# EPICS autosave request: iocBoot/ioc13ida_linux/Galil_settings.req
file "CARS_32_motor_settings.req",     P=$(P)
file "CARS_32_motor_positions.req",    P=$(P)
file "galil_8_motor_extras.req",       P=$(P)Galil1:, M1=m1,  M2=m2,  M3=m3,  M4=m4,  M5=m5,  M6=m6,  M7=m7,  M8=m8
file "galil_8_motor_extras.req",       P=$(P)Galil2:, M1=m9,  M2=m10, M3=m11, M4=m12, M5=m13, M6=m14, M7=m15, M8=m16
file "galil_8_motor_extras.req",       P=$(P)Galil3:, M1=m17, M2=m18, M3=m19, M4=m20, M5=m21, M6=m22, M7=m23, M8=m24
file "galil_8_motor_extras.req",       P=$(P)Galil4:, M1=m25, M2=m26, M3=m27, M4=m28, M5=m29, M6=m30, M7=m31, M8=m32
